PROGRAM AxisTestProg
VAR
    limitsPower AT %Q*: BOOL :=TRUE;
END_VAR

astAxes[1].stControl.bEnable:= TRUE;

END_PROGRAM

(* stored: Version 1.1.0.1, ProductVersion 3.1.4024.11
   POU AxisTestProg: Id {bde0c31b-9af8-4eb7-ac0d-a1bf58e721b3}, SpecialFunc None *)
